FUNCTION_BLOCK AD_TO_AR (* Composite FB for converting AD (DWORD) adapter to AR (REAL) adapter — ⚠ BIT-REINTERPRETATION, NOT a numeric cast! A raw counter/analog value is misinterpreted as IEEE754 bits. See AD_TO_AR_TODO.md / AD_TO_AR_NUM for the safe two-stage (bit-string->int->real) alternative. *)
  (* Standard: 61499-2; Description: Copyright (c) 2026 HR Agrartechnik GmbH This program and the accompanying materials are made available under the terms of the Eclipse Public License 2.0 which is available at https://www.eclipse.org/legal/epl-2.0/ SPDX-License-Identifier: EPL-2.0 *)
  (* Version 1.0, 2026-02-17, Franz Höpfinger, HR Agrartechnik GmbH *)
  PACKAGE adapter::conversion::unidirectional;
  (* Documentation:
  AD_TO_AR
   🇩🇪 Deutsch
   ⚠️ Achtung: Dieser Baustein wandelt DWORD nicht numerisch in REAL um, sondern nutzt intern F_DWORD_TO_REAL, was im FORTE-Kern für Bit-String-Quelltypen (BYTE/WORD/DWORD/LWORD) eine reine IEEE754-Bit-Reinterpretation ist. Ein roher Zähler-/Analogwert wie DWORD#2048 wird dadurch NICHT zu REAL#2048.0, sondern zu einer bedeutungslosen Zahl nahe Null.
   AD_TO_AR ist trotzdem korrekt und sinnvoll, wenn AD_IN bereits ein Bitmuster ist, das als REAL interpretiert werden soll (z. B. das Ergebnis von F_REAL_TO_DWORD oder ein anderweitig serialisiertes Float).
   Für einen echten Zahlenwert (z. B. Analog-Rohwert, Zähler) siehe stattdessen AD_TO_AR_NUM im selben Ordner — gleiche Schnittstelle, aber numerisch korrekt (Kette DWORD→UDINT→REAL).
   🇬🇧 English
   ⚠️ Warning: This block does not numerically convert DWORD to REAL — it internally uses F_DWORD_TO_REAL, which in the FORTE core is a pure IEEE754 bit-reinterpretation for bit-string source types (BYTE/WORD/DWORD/LWORD). A raw counter/analog value such as DWORD#2048 will NOT become REAL#2048.0, but a meaningless value near zero.
   AD_TO_AR is still correct and useful when AD_IN is already a bit pattern meant to be interpreted as REAL (e.g. the result of F_REAL_TO_DWORD, or otherwise serialized float data).
   For an actual numeric value (e.g. raw analog value, counter), use AD_TO_AR_NUM in the same folder instead — same interface, but numerically correct (DWORD→UDINT→REAL chain).
  *)
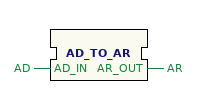
  SOCKETS
    AD_IN : adapter::types::unidirectional::AD; (* DWORD Adapter Input *)
  END_SOCKETS
  PLUGS
    AR_OUT : adapter::types::unidirectional::AR; (* REAL Adapter Output *)
  END_PLUGS
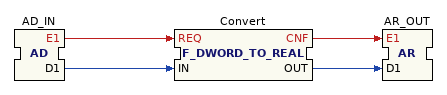
  FBS
    Convert : iec61131::conversion::F_DWORD_TO_REAL;
  END_FBS
  EVENT_CONNECTIONS
    AD_IN.E1 TO Convert.REQ;
    Convert.CNF TO AR_OUT.E1;
  END_CONNECTIONS
  DATA_CONNECTIONS
    AD_IN.D1 TO Convert.IN;
    Convert.OUT TO AR_OUT.D1;
  END_CONNECTIONS
END_FUNCTION_BLOCK
